% RSLogix 500 project MTRSTART_BAK000.RSS, saved by version 11.00.00.00 %
PROJECT "MTRSTART"    % processor: Bul.1763 MicroLogix 1100 Series A %

PROGRAM FILES
  LAD 2   2 rungs

DATA FILES
  O0 OUTPUT  4 elements
  I1 INPUT  6 elements
  S2 STATUS  66 elements
  B3 BINARY  1 elements
  T4 TIMER  1 elements
  C5 COUNTER  1 elements
  R6 CONTROL  1 elements
  N7 INTEGER  1 elements
  F8 FLOAT  1 elements

LADDER 2
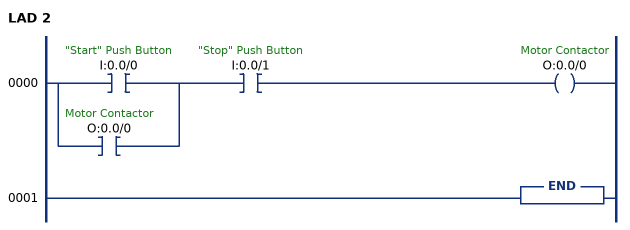
% Rung: 0 %
SOR BST XIC I:0.0/0 NXB XIC O:0.0/0 BND XIC I:0.0/1 OTE O:0.0/0 EOR
%   I:0.0/0  ""Start" Push Button" %
%   O:0.0/0  "Motor Contactor" %
%   I:0.0/1  ""Stop" Push Button" %
% Rung: 1 %
SOR END EOR
